// TwinCAT 3 PLC project StopWatch
// ProgramVersion: 3.1.4026.11
// CompilerDefines: VISU_USEPROPERTYINFO
// libraries:
//   Tc2_Standard, * (Beckhoff Automation GmbH)
//   Tc2_System, * (Beckhoff Automation GmbH)
//   Tc2_Utilities, * (Beckhoff Automation GmbH)
//   Tc3_Module, * (Beckhoff Automation GmbH)
//   VisuSymbols, 4.5.0.0 (System)
// project tree:
//   / GlobalTextList.TcGTLO, PlcTask.TcTTO (not stored), Visualization Manager.TcVMO (not stored)
//   POUs/ FB_FormatTime.TcPOU (not stored), FB_Interval.TcPOU (not stored), FB_Timer.TcPOU, MAIN.TcPOU (not stored)
//   VISUs/ Main_views.TcVIS
// real-time tasks:
//   TASK PlcTask: cycle T#10ms, priority 20, ADS port 350

// ---- POUs/FB_Timer.TcPOU
FUNCTION_BLOCK FB_Timer
VAR_INPUT
	bStart:BOOL;
	bPause:BOOL;
	bReset:BOOL;
	Starting: BOOL;
	Running: BOOL:=FALSE;
	
END_VAR
VAR_OUTPUT
	ElapsedTime:TIME:=T#0MS;
	
END_VAR
VAR
	bStartD: R_TRIG;
	
	
END_VAR

bStartD(CLK:=bStart);
IF bStartD.Q THEN
	Starting:=TRUE;
END_IF
IF bStart AND NOT Running THEN
	Running:=True;
	bStart:=FALSE;
		
ELSIF bReset THEN
	ElapsedTime:=T#0MS;
	bReset:=FALSE;	
	Running:=FALSE;
	
	
ELSIF bPause THEN
	Running:=FALSE;
	bPause:=FALSE;

END_IF
IF Running THEN 
	ElapsedTime:=Elapsedtime+T#10ms;
END_IF

END_FUNCTION_BLOCK

// ---- GlobalTextList.TcGTLO
TEXTLIST GlobalTextList
  37 = '%f'
  405 = '%s'
  659 = '%S'
  330 = 'h'
  266 = 'Interval'
  847 = 'INTERVALS'
  213 = 'LAP'
  723 = 'PAUSE'
  319 = 'R'
  890 = 'REET'
  585 = 'RESET'
  271 = 'S'
  694 = 'START'
  778 = 'StopWatch'
  36 = 'TimeView'
  880 = 'VIEW'
END_TEXTLIST

// ---- VISUs/Main_views.TcVIS
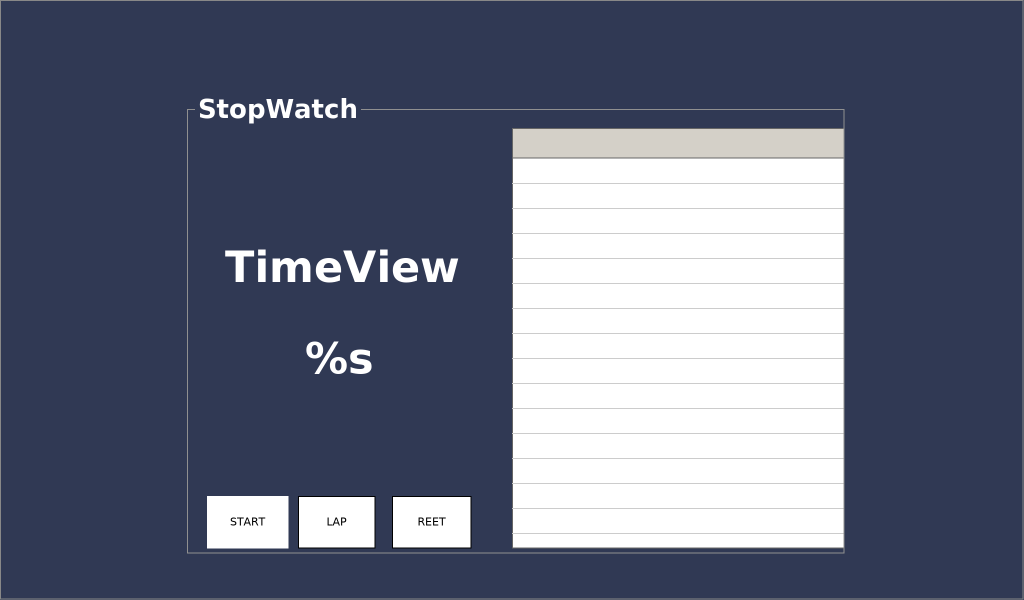
VISUALIZATION Main_views  // 1024x600
    Textfield (177,305 325x107), "%s", text variable: MAIN.FormattedTime
    Table (512,128 332x420), data array: MAIN.FormattedIntervals
        p3854506369: MAIN.FormattedIntervals[INDEX]
        p1014161805: 20 - 1 + INT#1
    Textfield (214,218 257x98), "TimeView"
    RoundedRectangle (207,496 81x52), "PAUSE", invisible if: NOT(MAIN.Timer.Running)
        tap MAIN.PauseButton
    RoundedRectangle (392,496 79x52), "REET"
        tap MAIN.ResetButton
    RoundedRectangle (298,496 77x52), "LAP", text variable: MAIN.IntervalButton
        tap MAIN.IntervalButton
    RoundedRectangle (207,496 81x52), "START", invisible if: MAIN.Timer.Running
        tap MAIN.StartButton
    Textfield (120,26 768x105)
    GroupBox (187,101 657x452), "StopWatch"
END_VISUALIZATION
